PROGRAM Axis01_Product_Position
VAR
	T1: TON;
//System_Bit
	Always_ON	:	BOOL	:=TRUE	;//상시 ON 
	Always_OFF	:	BOOL	:=FALSE	;//상시 OFF

END_VAR

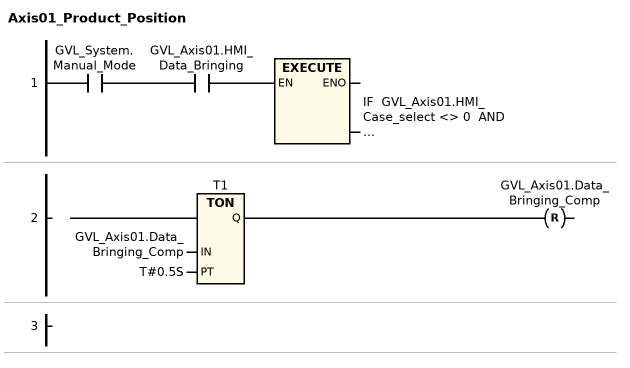
// NETWORK 1
IF GVL_System.Manual_Mode AND GVL_Axis01.HMI_Data_Bringing THEN
    IF  GVL_Axis01.HMI_Case_select <> 0	AND GVL_Axis01.HMI_Data_Bringing THEN
        GVL_Axis01.Selected_Position_Data := GVL_Axis01.Product_Position_Data[GVL_Axis01.HMI_Case_select];
        GVL_Axis01.Data_Bringing_Comp	:=	TRUE;
    END_IF
END_IF

// NETWORK 2
T1(IN := GVL_Axis01.Data_Bringing_Comp, PT := T#0.5S); // TON
GVL_Axis01.Data_Bringing_Comp R= T1.Q;

// NETWORK 3

END_PROGRAM

(* stored: Version 1.1.0.1, ProductVersion 3.1.4024.15
   POU Axis01_Product_Position: Id {c6a3b9f5-e248-4b6b-bb4b-7642bf686bd6}, SpecialFunc None *)
